// LS Electric XG5000 project: 0122 PLC incp, decp
// PLC LSPLC

PROGRAM NewProgram (task: 스캔 프로그램)

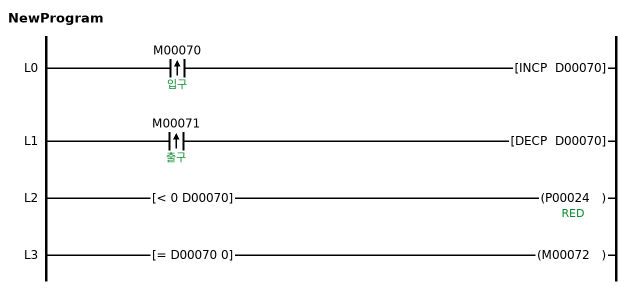
; L0
LOADP     M00070	// 입구
INCP      D00070
; L1
LOADP     M00071	// 출구
DECP      D00070
; L2
LOAD<     0 D00070
OUT       P00024	// RED
; L3
LOAD=     D00070 0
OUT       M00072

VARIABLES AND COMMENTS (devices not used above)
M00010	BIT	스위치 1
D00000	WORD	전번
M00001	BIT	스위치2
D00022	WORD	현재카운터수
M00002	BIT	스위치3
M00003	BIT	카운터
M00004	BIT	카운터 리셋
C0000	BIT/WORD	카운트
M00000	BIT	스위치1
M00041	BIT	더하기
D00030	WORD	입력1
D00032	WORD	입력2
D00040	WORD	결과
M00042	BIT	빼기
M00043	BIT	곱하기
M00044	BIT	나누기
M00045	BIT	CLR
M00060	BIT	운전
T0000	BIT/WORD	시간
P00025	BIT	YELLOW
M00090	BIT	P24
M00091	BIT	P25
M00092	BIT	GREEN
P00026	BIT	GREEN
M00100	BIT	wk
D00100	WORD	sec
D00101	WORD	인원
M00200	BIT	0이상